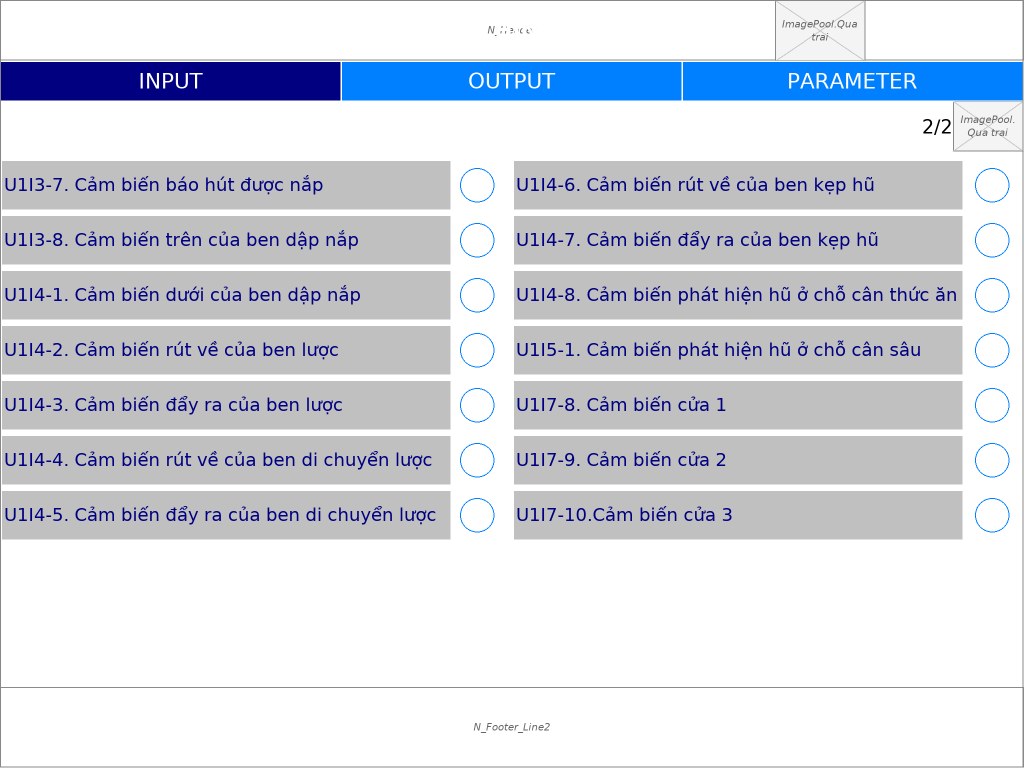
VISUALIZATION N_PLC_I2_next  // 1024x768
    Rectangle (886,102 103x50), "2/2"
    Frame (0,687 1024x80)
        shows N_Footer_Line2()
    Frame (0,0 1024x60)
        shows N_Header()
    Textfield (353,5 400x50), "MÀN HÌNH IO LINE 2"
    Image (775,0 90x61), image: ImagePool.Qua trai
        OnMouseClick: change screen: N_PLC_I2
    Rectangle (1,160 450x50), "U1I3-7. Cảm biến báo hút được nắp"
    Rectangle (1,215 450x50), "U1I3-8. Cảm biến trên của ben dập nắp"
    Rectangle (1,325 450x50), "U1I4-2. Cảm biến rút về của ben lược"
    Rectangle (1,270 450x50), "U1I4-1. Cảm biến dưới của ben dập nắp"
    Rectangle (1,380 450x50), "U1I4-3. Cảm biến đẩy ra của ben lược"
    Rectangle (1,435 450x50), "U1I4-4. Cảm biến rút về của ben di chuyển lược"
    Rectangle (1,490 450x50), "U1I4-5. Cảm biến đẩy ra của ben di chuyển lược"
    Ellipse (460,168 34x34), colour toggle: PR_Line02.fb_LidSupply.fbLidSuctionValve.bPressure, input disabled if: true
    Ellipse (460,223 34x34), colour toggle: PR_Line02.fb_LidClose.fbCylinder_LidClose.bAtRetract, input disabled if: true
    Ellipse (460,278 34x34), colour toggle: PR_Line02.fb_LidClose.fbCylinder_LidClose.bAtExtend, input disabled if: true
    Ellipse (460,333 34x34), colour toggle: PR_Line02.fb_Transfer.fbCylinder_Comb.bAtRetract, input disabled if: true
    Ellipse (460,388 34x34), colour toggle: PR_Line02.fb_Transfer.fbCylinder_Comb.bAtExtend, input disabled if: true
    Ellipse (460,443 34x34), colour toggle: PR_Line02.fb_Transfer.fbCylinder_Move_Comb.bAtRetract, input disabled if: true
    Ellipse (460,498 34x34), colour toggle: PR_Line02.fb_Transfer.fbCylinder_Move_Comb.bAtExtend, input disabled if: true
    Rectangle (513,215 450x50), "U1I4-7. Cảm biến đẩy ra của ben kẹp hũ"
    Rectangle (513,160 450x50), "U1I4-6. Cảm biến rút về của ben kẹp hũ"
    Rectangle (513,270 450x50), "U1I4-8. Cảm biến phát hiện hũ ở chỗ cân thức ăn"
    Rectangle (513,325 450x50), "U1I5-1. Cảm biến phát hiện hũ ở chỗ cân sâu"
    Rectangle (513,380 450x50), "U1I7-8. Cảm biến cửa 1"
    Rectangle (513,435 450x50), "U1I7-9. Cảm biến cửa 2"
    Rectangle (513,490 450x50), "U1I7-10.Cảm biến cửa 3"
    Ellipse (975,168 34x34), colour toggle: PR_Line02.fb_Transfer.fbCylinder_Clip.bAtRetract, input disabled if: true
    Ellipse (975,223 34x34), colour toggle: PR_Line02.fb_Transfer.fbCylinder_Clip.bAtRetract, input disabled if: true
    Ellipse (975,278 34x34), colour toggle: PR_Line02.fb_FoodWeight.bCupPresent, input disabled if: true
    Ellipse (975,333 34x34), colour toggle: PR_Line02.fb_WormWeight.bCupPresent, input disabled if: true
    Ellipse (975,388 34x34), colour toggle: GVL_IO.bSafetyDoor1, input disabled if: true
    Ellipse (975,443 34x34), colour toggle: GVL_IO.bSafetyDoor2, input disabled if: true
    Ellipse (975,498 34x34), colour toggle: GVL_IO.bSafetyDoor3, input disabled if: true
    Image (953,101 70x50), image: ImagePool.Qua trai
        OnMouseClick: change screen: N_PLC_I2
    Rectangle (0,61 341x40), "INPUT"
        OnMouseClick: change screen: N_PLC_I2
    Rectangle (341,61 341x40), "OUTPUT"
        OnMouseClick: change screen: N_PLC_O2
    Rectangle (682,61 341x40), "PARAMETER"
        OnMouseClick: change screen: N_Parameter_2
END_VISUALIZATION

(* stored: Version 1.1.0.1, ProductVersion 3.1.4024.12
   Visu N_PLC_I2_next: Id {1b8a118c-5a1d-458f-9000-7fe40510bcda} *)
